// TIA Portal project "Project1" (V15)

(* hardware
DEVICE "S7-1200 station_1"  S7-1200 Station
   slot 0: "Rack_0"  S7-1200 Rack  Rack  V1.0
   slot 1: "PLC_1"  CPU 1214C DC/DC/DC  6ES7 214-1AG40-0XB0  V4.2
DEVICE "HMI_1"  TP1500 Basic color PN
   slot 0: "HMI_1"  TP1500 Basic color PN  6AV6 647-0AG11-3AX0  12.0.0.0
   slot 1: "HMI_RT_1"  TP1500 Basic color PN  6AV6 647-0AG11-3AX0  12.0.0.0
   slot 5: "HMI_1.IE_CP_1"  PROFINET Interface  12.0.0.0
      slot 1: "PROFINET Interface_1"  PROFINET Interface
         slot 1: "Port_1"  Port
*)

// ===== PLC "PLC_1"  CPU 1214C DC/DC/DC =====

VAR_GLOBAL   // PLC tag table "Default tag table"
   "btn_Start" AT %M9.0 : Bool;
   "Program_RUN" AT %M10.0 : Bool;
   "btn_Stop" AT %M9.1 : Bool;
   "SS_NG" AT %M11.0 : Bool;
   "M_NG" AT %M10.1 : Bool;
   "ok_add" AT %M10.2 : Bool;
   "ok_delete" AT %M10.3 : Bool;
   "SS_input" AT %M11.1 : Bool;
   "SS_output" AT %M11.2 : Bool;
   "Reject" AT %Q1.0 : Bool;
   "Process_1" AT %M12.0 : Bool;
   "Process_2" AT %M12.1 : Bool;
   "Process_3" AT %M12.2 : Bool;
   "Process_4" AT %M12.3 : Bool;
   "Process_5" AT %M12.4 : Bool;
   "Process_6" AT %M12.5 : Bool;
   "Process_7" AT %M12.6 : Bool;
   "Process_8" AT %M12.7 : Bool;
   "ok_P1" AT %M13.0 : Bool;
   "ok_P2" AT %M13.1 : Bool;
   "ok_P3" AT %M13.2 : Bool;
   "ok_P4" AT %M13.3 : Bool;
   "ok_P5" AT %M13.4 : Bool;
   "ok_P6" AT %M13.5 : Bool;
   "ok_P7" AT %M13.6 : Bool;
   "ok_P8" AT %M13.7 : Bool;
   "Process" AT %MB12 : Byte;
   "ok_shift" AT %M10.4 : Bool;
   "M_cnt" AT %M10.5 : Bool;
   "ok_shifttttt" AT %M10.6 : Bool;
END_VAR

DATA_BLOCK "Data_HERE"   // DB1
{ S7_Optimized_Access := 'TRUE' }
VERSION : 0.1
   VAR
      "step" : Byte := 2#00000001;
      count_1 : Int := 0;
      count_2 : Int := 0;
      count_3 : Int := 0;
      count_4 : Int := 0;
      count_5 : Int := 0;
      count_6 : Int := 0;
      count_7 : Int := 0;
      count_8 : Int := 0;
   END_VAR
BEGIN
END_DATA_BLOCK

// folder: System blocks/Program resources

DATA_BLOCK "IEC_Counter_1"   // DB2
{ S7_Optimized_Access := 'TRUE' }
AUTHOR : Simatic
FAMILY : IEC
NAME : CNTR
VERSION : 1.0
// stored: InstanceOfName IEC_COUNTER
"IEC_COUNTER"
BEGIN
END_DATA_BLOCK

DATA_BLOCK "IEC_Timer_Process_1"   // DB3
{ S7_Optimized_Access := 'TRUE' }
AUTHOR : Simatic
FAMILY : IEC
NAME : IEC_TMR
VERSION : 1.0
// stored: InstanceOfName IEC_TIMER
"IEC_TIMER"
BEGIN
END_DATA_BLOCK

DATA_BLOCK "IEC_Timer_Process_2"   // DB4
{ S7_Optimized_Access := 'TRUE' }
AUTHOR : Simatic
FAMILY : IEC
NAME : IEC_TMR
VERSION : 1.0
// stored: InstanceOfName IEC_TIMER
"IEC_TIMER"
BEGIN
END_DATA_BLOCK

DATA_BLOCK "IEC_Timer_Process_3"   // DB5
{ S7_Optimized_Access := 'TRUE' }
AUTHOR : Simatic
FAMILY : IEC
NAME : IEC_TMR
VERSION : 1.0
// stored: InstanceOfName IEC_TIMER
"IEC_TIMER"
BEGIN
END_DATA_BLOCK

DATA_BLOCK "IEC_Timer_Process_4"   // DB6
{ S7_Optimized_Access := 'TRUE' }
AUTHOR : Simatic
FAMILY : IEC
NAME : IEC_TMR
VERSION : 1.0
// stored: InstanceOfName IEC_TIMER
"IEC_TIMER"
BEGIN
END_DATA_BLOCK

DATA_BLOCK "IEC_Timer_Process_5"   // DB7
{ S7_Optimized_Access := 'TRUE' }
AUTHOR : Simatic
FAMILY : IEC
NAME : IEC_TMR
VERSION : 1.0
// stored: InstanceOfName IEC_TIMER
"IEC_TIMER"
BEGIN
END_DATA_BLOCK

DATA_BLOCK "IEC_Timer_Process_6"   // DB8
{ S7_Optimized_Access := 'TRUE' }
AUTHOR : Simatic
FAMILY : IEC
NAME : IEC_TMR
VERSION : 1.0
// stored: InstanceOfName IEC_TIMER
"IEC_TIMER"
BEGIN
END_DATA_BLOCK

DATA_BLOCK "IEC_Timer_Process_7"   // DB9
{ S7_Optimized_Access := 'TRUE' }
AUTHOR : Simatic
FAMILY : IEC
NAME : IEC_TMR
VERSION : 1.0
// stored: InstanceOfName IEC_TIMER
"IEC_TIMER"
BEGIN
END_DATA_BLOCK

DATA_BLOCK "IEC_Timer_Process_8"   // DB10
{ S7_Optimized_Access := 'TRUE' }
AUTHOR : Simatic
FAMILY : IEC
NAME : IEC_TMR
VERSION : 1.0
// stored: InstanceOfName IEC_TIMER
"IEC_TIMER"
BEGIN
END_DATA_BLOCK

DATA_BLOCK "IEC_Timer_shift"   // DB11
{ S7_Optimized_Access := 'TRUE' }
AUTHOR : Simatic
FAMILY : IEC
NAME : IEC_TMR
VERSION : 1.0
// stored: InstanceOfName IEC_TIMER
"IEC_TIMER"
BEGIN
END_DATA_BLOCK

// folder: (top level)

FUNCTION "SystemReject" : Void   // FC1, LAD
{ S7_Optimized_Access := 'TRUE' }
VERSION : 0.1
BEGIN

REGION Network 1
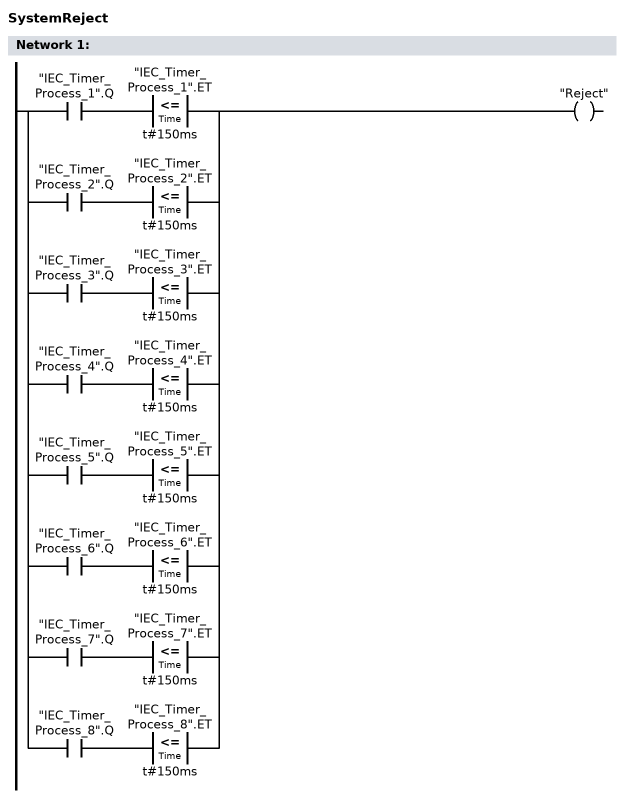
   RUNG wire#powerrail
      Contact( "IEC_Timer_Process_1".Q )
      { S7_Templates := "SrcType := Time" } LE_Contact(in1 := "IEC_Timer_Process_1".ET, in2 := t#150ms)
      wire#w1
      Coil( "Reject" )
   END_RUNG
   RUNG wire#powerrail
      Contact( "IEC_Timer_Process_2".Q )
      { S7_Templates := "SrcType := Time" } LE_Contact(in1 := "IEC_Timer_Process_2".ET, in2 := t#150ms)
   END_RUNG wire#w1
   RUNG wire#powerrail
      Contact( "IEC_Timer_Process_3".Q )
      { S7_Templates := "SrcType := Time" } LE_Contact(in1 := "IEC_Timer_Process_3".ET, in2 := t#150ms)
   END_RUNG wire#w1
   RUNG wire#powerrail
      Contact( "IEC_Timer_Process_4".Q )
      { S7_Templates := "SrcType := Time" } LE_Contact(in1 := "IEC_Timer_Process_4".ET, in2 := t#150ms)
   END_RUNG wire#w1
   RUNG wire#powerrail
      Contact( "IEC_Timer_Process_5".Q )
      { S7_Templates := "SrcType := Time" } LE_Contact(in1 := "IEC_Timer_Process_5".ET, in2 := t#150ms)
   END_RUNG wire#w1
   RUNG wire#powerrail
      Contact( "IEC_Timer_Process_6".Q )
      { S7_Templates := "SrcType := Time" } LE_Contact(in1 := "IEC_Timer_Process_6".ET, in2 := t#150ms)
   END_RUNG wire#w1
   RUNG wire#powerrail
      Contact( "IEC_Timer_Process_7".Q )
      { S7_Templates := "SrcType := Time" } LE_Contact(in1 := "IEC_Timer_Process_7".ET, in2 := t#150ms)
   END_RUNG wire#w1
   RUNG wire#powerrail
      Contact( "IEC_Timer_Process_8".Q )
      { S7_Templates := "SrcType := Time" } LE_Contact(in1 := "IEC_Timer_Process_8".ET, in2 := t#150ms)
   END_RUNG wire#w1
   // the same network as SCL:
   "Reject" := ("IEC_Timer_Process_1".Q AND ("IEC_Timer_Process_1".ET <= t#150ms)) OR ("IEC_Timer_Process_2".Q AND ("IEC_Timer_Process_2".ET <= t#150ms)) OR ("IEC_Timer_Process_3".Q AND ("IEC_Timer_Process_3".ET <= t#150ms)) OR ("IEC_Timer_Process_4".Q AND ("IEC_Timer_Process_4".ET <= t#150ms)) OR ("IEC_Timer_Process_5".Q AND ("IEC_Timer_Process_5".ET <= t#150ms)) OR ("IEC_Timer_Process_6".Q AND ("IEC_Timer_Process_6".ET <= t#150ms)) OR ("IEC_Timer_Process_7".Q AND ("IEC_Timer_Process_7".ET <= t#150ms)) OR ("IEC_Timer_Process_8".Q AND ("IEC_Timer_Process_8".ET <= t#150ms));
END_REGION
END_FUNCTION

FUNCTION "SystemShift" : Void   // FC2, LAD
{ S7_Optimized_Access := 'TRUE' }
VERSION : 0.1
   VAR_TEMP   // added for the SCL form of the ladder/FBD networks
      _w1 : Bool;
      _w2 : Bool;
   END_VAR
BEGIN

REGION Network 1
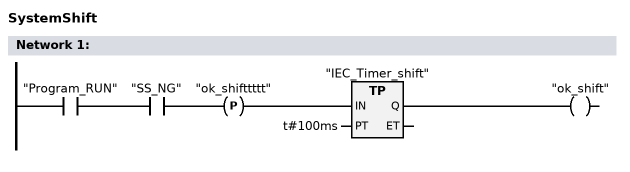
   #_w1 := "Program_RUN" AND "SS_NG";
   #_w2 := #_w1 AND NOT "ok_shifttttt";   // rising edge
   "ok_shifttttt" := #_w1;
   "IEC_Timer_shift".TP(IN := #_w2, PT := t#100ms);
   "ok_shift" := "IEC_Timer_shift".Q;
END_REGION
END_FUNCTION

FUNCTION "SystemReset" : Void   // FC3, LAD
{ S7_Optimized_Access := 'TRUE' }
VERSION : 0.1
BEGIN

REGION Network 1
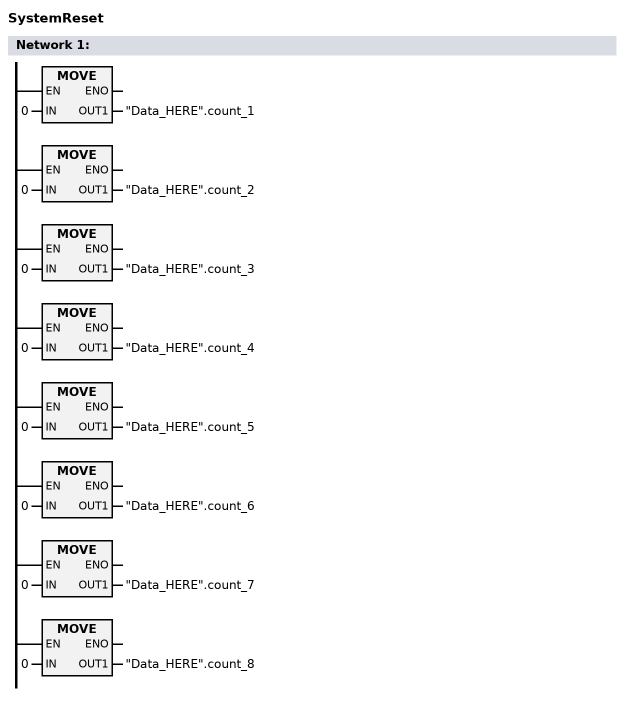
   RUNG wire#powerrail
      Move(in := 0, out1 => "Data_HERE".count_1)
   END_RUNG
   RUNG wire#powerrail
      Move(in := 0, out1 => "Data_HERE".count_2)
   END_RUNG
   RUNG wire#powerrail
      Move(in := 0, out1 => "Data_HERE".count_3)
   END_RUNG
   RUNG wire#powerrail
      Move(in := 0, out1 => "Data_HERE".count_4)
   END_RUNG
   RUNG wire#powerrail
      Move(in := 0, out1 => "Data_HERE".count_5)
   END_RUNG
   RUNG wire#powerrail
      Move(in := 0, out1 => "Data_HERE".count_6)
   END_RUNG
   RUNG wire#powerrail
      Move(in := 0, out1 => "Data_HERE".count_7)
   END_RUNG
   RUNG wire#powerrail
      Move(in := 0, out1 => "Data_HERE".count_8)
   END_RUNG
   // the same network as SCL:
   "Data_HERE".count_1 := 0;
   "Data_HERE".count_2 := 0;
   "Data_HERE".count_3 := 0;
   "Data_HERE".count_4 := 0;
   "Data_HERE".count_5 := 0;
   "Data_HERE".count_6 := 0;
   "Data_HERE".count_7 := 0;
   "Data_HERE".count_8 := 0;
END_REGION
END_FUNCTION

ORGANIZATION_BLOCK "Main"   // OB1, LAD, ProgramCycle
TITLE = "Main Program Sweep (Cycle)"
{ S7_Optimized_Access := 'TRUE' }
VERSION : 0.1
   VAR_INPUT
      Initial_Call : Bool;   // Initial call of this OB
      Remanence : Bool;   // =True, if remanent data are available
   END_VAR
   VAR_TEMP   // added for the SCL form of the ladder/FBD networks
      _w1 : Bool;
      _w2 : Bool;
      _w3 : Bool;
      _w4 : Bool;
   END_VAR
BEGIN

REGION Network 1: Start / Stop
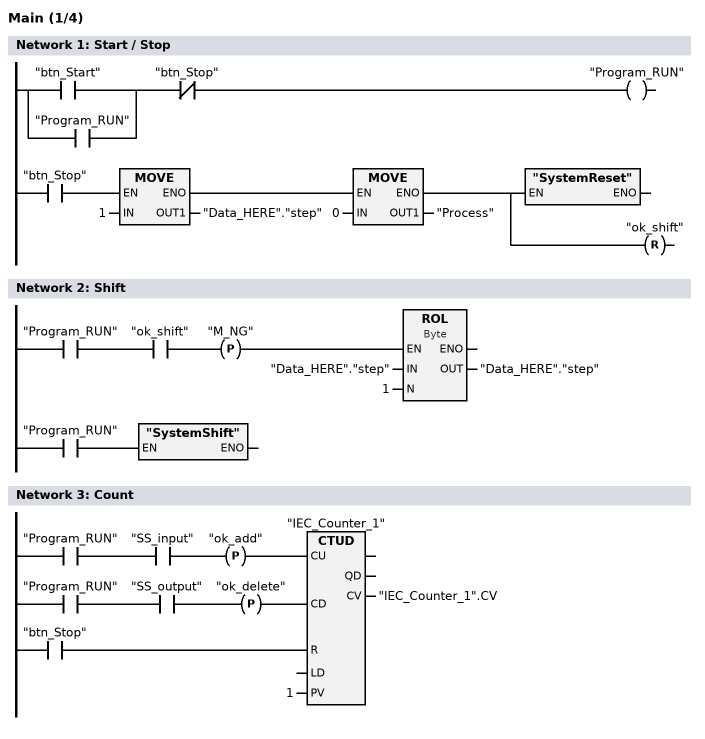
   RUNG wire#powerrail
      Contact( "btn_Start" )
      wire#w1
      I_Contact( "btn_Stop" )
      Coil( "Program_RUN" )
   END_RUNG
   RUNG wire#powerrail
      Contact( "Program_RUN" )
   END_RUNG wire#w1
   RUNG wire#powerrail
      Contact( "btn_Stop" )
      Move(in := 1, out1 => "Data_HERE"."step")
      Move(in := 0, out1 => "Process")
      wire#w2
      "SystemReset"()
   END_RUNG
   RUNG wire#w2
      R_Coil( "ok_shift" )
   END_RUNG
   // the same network as SCL:
   "Program_RUN" := ("btn_Start" OR "Program_RUN") AND NOT "btn_Stop";
   IF "btn_Stop" THEN
       "Data_HERE"."step" := 1;
       "Process" := 0;
   END_IF;
   #_w1 := "btn_Stop";
   IF #_w1 THEN
       "SystemReset"();
       "ok_shift" := FALSE;
   END_IF;
END_REGION

REGION Network 2: Shift
   #_w1 := "Program_RUN" AND "ok_shift";
   #_w2 := #_w1 AND NOT "M_NG";   // rising edge
   "M_NG" := #_w1;
   IF #_w2 THEN "Data_HERE"."step" := ROL(IN := "Data_HERE"."step", N := 1); END_IF;
   IF "Program_RUN" THEN "SystemShift"(); END_IF;
END_REGION

REGION Network 3: Count
   #_w1 := "Program_RUN" AND "SS_input";
   #_w2 := #_w1 AND NOT "ok_add";   // rising edge
   "ok_add" := #_w1;
   #_w3 := "Program_RUN" AND "SS_output";
   #_w4 := #_w3 AND NOT "ok_delete";   // rising edge
   "ok_delete" := #_w3;
   "IEC_Counter_1".CTUD(CU := #_w2, CD := #_w4, R := "btn_Stop", PV := 1, CV => "IEC_Counter_1".CV);
END_REGION

REGION Network 4: Loop Triger NG
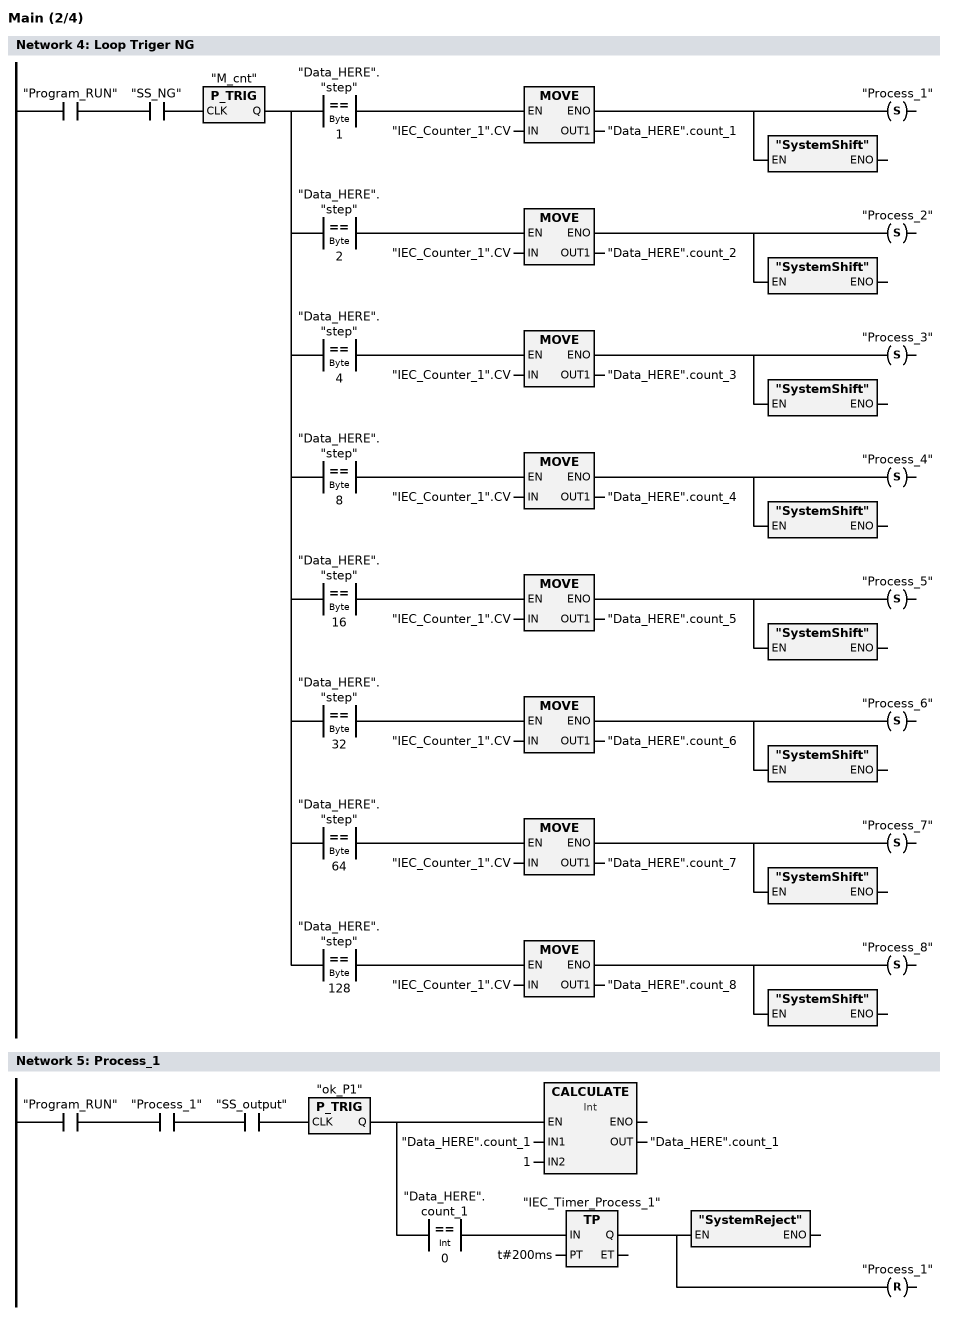
   RUNG wire#powerrail
      Contact( "Program_RUN" )
      Contact( "SS_NG" )
      P_Trig( "M_cnt" )
      wire#w1
      { S7_Templates := "SrcType := Byte" } EQ_Contact(in1 := "Data_HERE"."step", in2 := 1)
      Move(in := "IEC_Counter_1".CV, out1 => "Data_HERE".count_1)
      wire#w2
      S_Coil( "Process_1" )
   END_RUNG
   RUNG wire#w2
      "SystemShift"()
   END_RUNG
   RUNG wire#w1
      { S7_Templates := "SrcType := Byte" } EQ_Contact(in1 := "Data_HERE"."step", in2 := 2)
      Move(in := "IEC_Counter_1".CV, out1 => "Data_HERE".count_2)
      wire#w3
      S_Coil( "Process_2" )
   END_RUNG
   RUNG wire#w3
      "SystemShift"()
   END_RUNG
   RUNG wire#w1
      { S7_Templates := "SrcType := Byte" } EQ_Contact(in1 := "Data_HERE"."step", in2 := 4)
      Move(in := "IEC_Counter_1".CV, out1 => "Data_HERE".count_3)
      wire#w4
      S_Coil( "Process_3" )
   END_RUNG
   RUNG wire#w4
      "SystemShift"()
   END_RUNG
   RUNG wire#w1
      { S7_Templates := "SrcType := Byte" } EQ_Contact(in1 := "Data_HERE"."step", in2 := 8)
      Move(in := "IEC_Counter_1".CV, out1 => "Data_HERE".count_4)
      wire#w5
      S_Coil( "Process_4" )
   END_RUNG
   RUNG wire#w5
      "SystemShift"()
   END_RUNG
   RUNG wire#w1
      { S7_Templates := "SrcType := Byte" } EQ_Contact(in1 := "Data_HERE"."step", in2 := 16)
      Move(in := "IEC_Counter_1".CV, out1 => "Data_HERE".count_5)
      wire#w6
      S_Coil( "Process_5" )
   END_RUNG
   RUNG wire#w6
      "SystemShift"()
   END_RUNG
   RUNG wire#w1
      { S7_Templates := "SrcType := Byte" } EQ_Contact(in1 := "Data_HERE"."step", in2 := 32)
      Move(in := "IEC_Counter_1".CV, out1 => "Data_HERE".count_6)
      wire#w7
      S_Coil( "Process_6" )
   END_RUNG
   RUNG wire#w7
      "SystemShift"()
   END_RUNG
   RUNG wire#w1
      { S7_Templates := "SrcType := Byte" } EQ_Contact(in1 := "Data_HERE"."step", in2 := 64)
      Move(in := "IEC_Counter_1".CV, out1 => "Data_HERE".count_7)
      wire#w8
      S_Coil( "Process_7" )
   END_RUNG
   RUNG wire#w8
      "SystemShift"()
   END_RUNG
   RUNG wire#w1
      { S7_Templates := "SrcType := Byte" } EQ_Contact(in1 := "Data_HERE"."step", in2 := 128)
      Move(in := "IEC_Counter_1".CV, out1 => "Data_HERE".count_8)
      wire#w9
      S_Coil( "Process_8" )
   END_RUNG
   RUNG wire#w9
      "SystemShift"()
   END_RUNG
   // the same network as SCL:
   #_w1 := "Program_RUN" AND "SS_NG";
   #_w2 := #_w1 AND NOT "M_cnt";   // rising edge
   "M_cnt" := #_w1;
   IF #_w2 AND ("Data_HERE"."step" = 1) THEN
       "Data_HERE".count_1 := "IEC_Counter_1".CV;
       "Process_1" := TRUE;
       "SystemShift"();
   END_IF;
   IF #_w2 AND ("Data_HERE"."step" = 2) THEN
       "Data_HERE".count_2 := "IEC_Counter_1".CV;
       "Process_2" := TRUE;
       "SystemShift"();
   END_IF;
   IF #_w2 AND ("Data_HERE"."step" = 4) THEN
       "Data_HERE".count_3 := "IEC_Counter_1".CV;
       "Process_3" := TRUE;
       "SystemShift"();
   END_IF;
   IF #_w2 AND ("Data_HERE"."step" = 8) THEN
       "Data_HERE".count_4 := "IEC_Counter_1".CV;
       "Process_4" := TRUE;
       "SystemShift"();
   END_IF;
   IF #_w2 AND ("Data_HERE"."step" = 16) THEN
       "Data_HERE".count_5 := "IEC_Counter_1".CV;
       "Process_5" := TRUE;
       "SystemShift"();
   END_IF;
   IF #_w2 AND ("Data_HERE"."step" = 32) THEN
       "Data_HERE".count_6 := "IEC_Counter_1".CV;
       "Process_6" := TRUE;
       "SystemShift"();
   END_IF;
   IF #_w2 AND ("Data_HERE"."step" = 64) THEN
       "Data_HERE".count_7 := "IEC_Counter_1".CV;
       "Process_7" := TRUE;
       "SystemShift"();
   END_IF;
   IF #_w2 AND ("Data_HERE"."step" = 128) THEN
       "Data_HERE".count_8 := "IEC_Counter_1".CV;
       "Process_8" := TRUE;
       "SystemShift"();
   END_IF;
END_REGION

REGION Network 5: Process_1
   #_w1 := "Program_RUN" AND "Process_1" AND "SS_output";
   #_w2 := #_w1 AND NOT "ok_P1";   // rising edge
   "ok_P1" := #_w1;
   IF #_w2 THEN "Data_HERE".count_1 := "Data_HERE".count_1-1; END_IF;
   "IEC_Timer_Process_1".TP(IN := #_w2 AND ("Data_HERE".count_1 = 0), PT := t#200ms);
   #_w3 := "IEC_Timer_Process_1".Q;
   IF #_w3 THEN
       "SystemReject"();
       "Process_1" := FALSE;
   END_IF;
END_REGION

REGION Network 6: Process_2
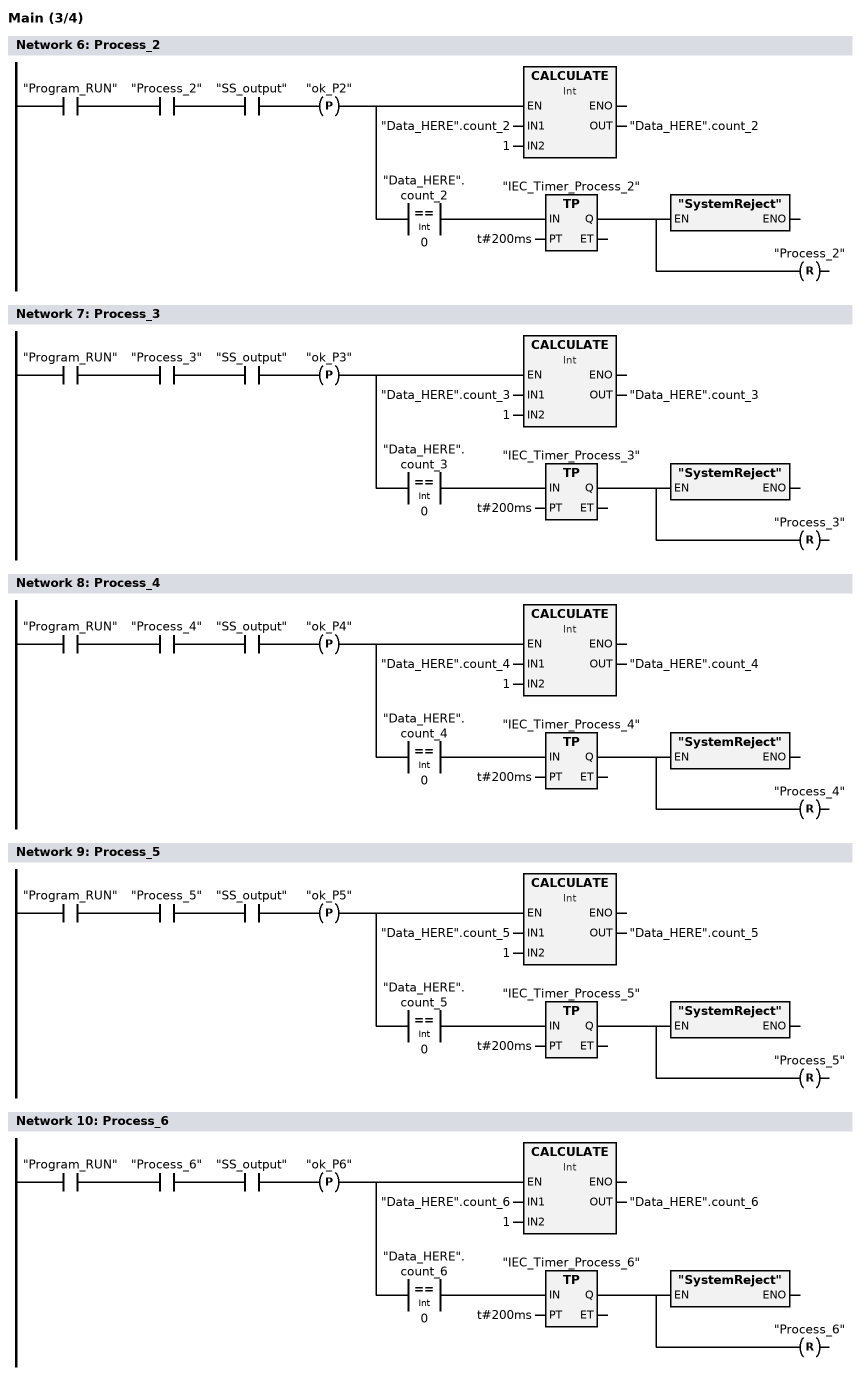
   #_w1 := "Program_RUN" AND "Process_2" AND "SS_output";
   #_w2 := #_w1 AND NOT "ok_P2";   // rising edge
   "ok_P2" := #_w1;
   IF #_w2 THEN "Data_HERE".count_2 := "Data_HERE".count_2-1; END_IF;
   "IEC_Timer_Process_2".TP(IN := #_w2 AND ("Data_HERE".count_2 = 0), PT := t#200ms);
   #_w3 := "IEC_Timer_Process_2".Q;
   IF #_w3 THEN
       "SystemReject"();
       "Process_2" := FALSE;
   END_IF;
END_REGION

REGION Network 7: Process_3
   #_w1 := "Program_RUN" AND "Process_3" AND "SS_output";
   #_w2 := #_w1 AND NOT "ok_P3";   // rising edge
   "ok_P3" := #_w1;
   IF #_w2 THEN "Data_HERE".count_3 := "Data_HERE".count_3-1; END_IF;
   "IEC_Timer_Process_3".TP(IN := #_w2 AND ("Data_HERE".count_3 = 0), PT := t#200ms);
   #_w3 := "IEC_Timer_Process_3".Q;
   IF #_w3 THEN
       "SystemReject"();
       "Process_3" := FALSE;
   END_IF;
END_REGION

REGION Network 8: Process_4
   #_w1 := "Program_RUN" AND "Process_4" AND "SS_output";
   #_w2 := #_w1 AND NOT "ok_P4";   // rising edge
   "ok_P4" := #_w1;
   IF #_w2 THEN "Data_HERE".count_4 := "Data_HERE".count_4-1; END_IF;
   "IEC_Timer_Process_4".TP(IN := #_w2 AND ("Data_HERE".count_4 = 0), PT := t#200ms);
   #_w3 := "IEC_Timer_Process_4".Q;
   IF #_w3 THEN
       "SystemReject"();
       "Process_4" := FALSE;
   END_IF;
END_REGION

REGION Network 9: Process_5
   #_w1 := "Program_RUN" AND "Process_5" AND "SS_output";
   #_w2 := #_w1 AND NOT "ok_P5";   // rising edge
   "ok_P5" := #_w1;
   IF #_w2 THEN "Data_HERE".count_5 := "Data_HERE".count_5-1; END_IF;
   "IEC_Timer_Process_5".TP(IN := #_w2 AND ("Data_HERE".count_5 = 0), PT := t#200ms);
   #_w3 := "IEC_Timer_Process_5".Q;
   IF #_w3 THEN
       "SystemReject"();
       "Process_5" := FALSE;
   END_IF;
END_REGION

REGION Network 10: Process_6
   #_w1 := "Program_RUN" AND "Process_6" AND "SS_output";
   #_w2 := #_w1 AND NOT "ok_P6";   // rising edge
   "ok_P6" := #_w1;
   IF #_w2 THEN "Data_HERE".count_6 := "Data_HERE".count_6-1; END_IF;
   "IEC_Timer_Process_6".TP(IN := #_w2 AND ("Data_HERE".count_6 = 0), PT := t#200ms);
   #_w3 := "IEC_Timer_Process_6".Q;
   IF #_w3 THEN
       "SystemReject"();
       "Process_6" := FALSE;
   END_IF;
END_REGION

REGION Network 11: Process_7
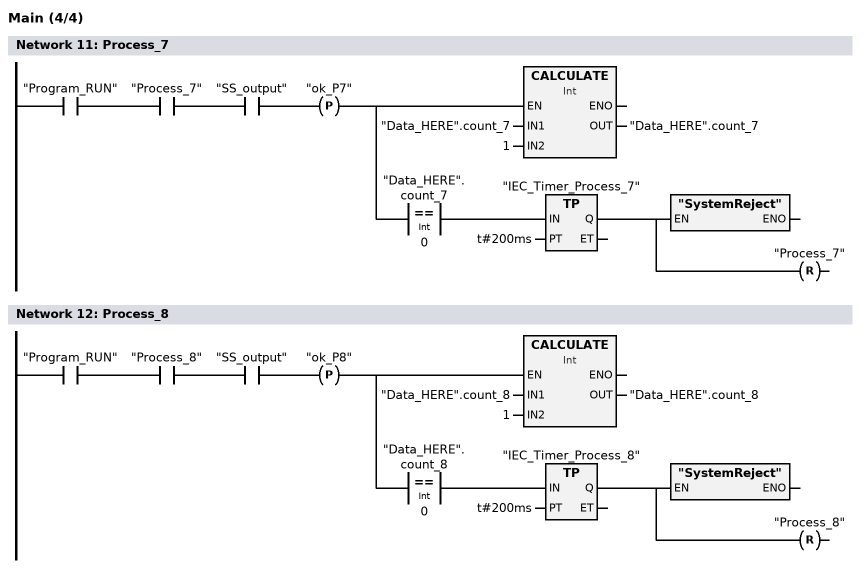
   #_w1 := "Program_RUN" AND "Process_7" AND "SS_output";
   #_w2 := #_w1 AND NOT "ok_P7";   // rising edge
   "ok_P7" := #_w1;
   IF #_w2 THEN "Data_HERE".count_7 := "Data_HERE".count_7-1; END_IF;
   "IEC_Timer_Process_7".TP(IN := #_w2 AND ("Data_HERE".count_7 = 0), PT := t#200ms);
   #_w3 := "IEC_Timer_Process_7".Q;
   IF #_w3 THEN
       "SystemReject"();
       "Process_7" := FALSE;
   END_IF;
END_REGION

REGION Network 12: Process_8
   #_w1 := "Program_RUN" AND "Process_8" AND "SS_output";
   #_w2 := #_w1 AND NOT "ok_P8";   // rising edge
   "ok_P8" := #_w1;
   IF #_w2 THEN "Data_HERE".count_8 := "Data_HERE".count_8-1; END_IF;
   "IEC_Timer_Process_8".TP(IN := #_w2 AND ("Data_HERE".count_8 = 0), PT := t#200ms);
   #_w3 := "IEC_Timer_Process_8".Q;
   IF #_w3 THEN
       "SystemReject"();
       "Process_8" := FALSE;
   END_IF;
END_REGION
END_ORGANIZATION_BLOCK

(* ===== HMI "HMI_RT_1" =====
system functions are stored by id; their names below are inferred from use
connection "HMI_Connection_1": ETHERNET, SMART_S7_1200_OMS

HMI tags "Default tag table"
   "btn_Start" : Bool = PLC btn_Start AT %M9.0, 100 ms
   "btn_Stop" : Bool = PLC btn_Stop AT %M9.1, 100 ms
   "SS_input" : Bool = PLC SS_input AT %M11.1, 100 ms
   "SS_output" : Bool = PLC SS_output AT %M11.2, 100 ms
   "SS_NG" : Bool = PLC SS_NG AT %M11.0, 100 ms
   "Reject" : Bool = PLC Reject AT %Q1.0, 100 ms

Template "Template_1" 1024x768
   Button "Exit" at 943,707 size 79x59; TextOff 'Exit'; PictureOff "ExitRuntime_TP1500_Basic_color_PN"; PictureOn "ExitRuntime_TP1500_Basic_color_PN"
      on Release: StopRuntime(0)
   Button "Template_Button" at 857,707 size 79x59; TextOff 'Text'
   Button "Template_Button_1" at 772,707 size 79x59; TextOff 'Text'
   Button "Template_Button_2" at 686,707 size 79x59; TextOff 'Text'
   Button "Template_Button_3" at 600,707 size 79x59; TextOff 'Text'
   Button "Template_Button_4" at 515,707 size 79x59; TextOff 'Text'
   Button "Template_Button_5" at 429,707 size 79x59; TextOff 'Text'
   Button "Template_Button_6" at 344,707 size 79x59; TextOff 'Text'
   Button "Template_Button_7" at 258,707 size 79x59; TextOff 'Text'
   Button "Template_Button_8" at 172,707 size 79x59; TextOff 'Text'
   Button "Alarms" at 87,707 size 79x59; TextOff 'Alarms'; PictureOff "AlarmDisplay_TP1500_Basic_color_PN"; PictureOn "AlarmDisplay_TP1500_Basic_color_PN"
      on Release: function_ef3f5d25("Alarm window_Unacknowledged", -1)
   Button "Start screen" at 1,707 size 79x59; TextOff 'Start screen'; PictureOff "NavigateHome_TP1500_Basic_color_PN"; PictureOn "NavigateHome_TP1500_Basic_color_PN"
      on Release: ActivateScreen("Root screen", 0)

screen "Root screen" 1024x768, template "Template_1"
   Button "HmiScreenItemData_1" at 36,36 size 159x47; TextOff 'System screens'; PictureOff "Navigates to System screens for TP1500 Basic color PN 12.0.0.0"; PictureOn "Navigates to System screens for TP1500 Basic color PN 12.0.0.0"
      on Release: ActivateScreen("System screens", 0)
   Button "Button_1" at 204,119 size 96x32; TextOff 'Start'
      on Press: SetBit("btn_Start")
      on Release: ResetBit("btn_Start")
   Button "Button_2" at 204,184 size 96x32; TextOff 'Stop'
      on Press: SetBit("btn_Stop")
      on Release: ResetBit("btn_Stop")
   Button "Button_3" at 54,117 size 96x32; TextOff 'INPUT'
      on Press: SetBit("SS_input")
      on Release: ResetBit("SS_input")
   Button "Button_4" at 50,178 size 96x32; TextOff 'OUTPUT'
      on Press: SetBit("SS_output")
      on Release: ResetBit("SS_output")
   Button "Button_5" at 54,244 size 96x32; TextOff 'NG'
      on Press: SetBit("SS_NG")
      on Release: ResetBit("SS_NG")
   Circle "Circle_1" at 218,244 size 48x48
      Appearance <- "Reject"

screen "System screens" 1024x768, template "Template_1"
   Button "Back" at 1,1 size 159x47; TextOff 'Back'
      on Release: ActivateScreen("Root screen", 0)
*)